Omron CX-Programmer project 新規ﾌﾟﾛｼﾞｪｸﾄ (CX-Programmer 9.61)

# PLC hoge1: CP1L L

## Program 新規ﾌﾟﾛｸﾞﾗﾑ1 (cyclic task 0)
Local symbols
I 0.00 BOOL
Q 100.00 BOOL

### Section ｾｸｼｮﾝ1

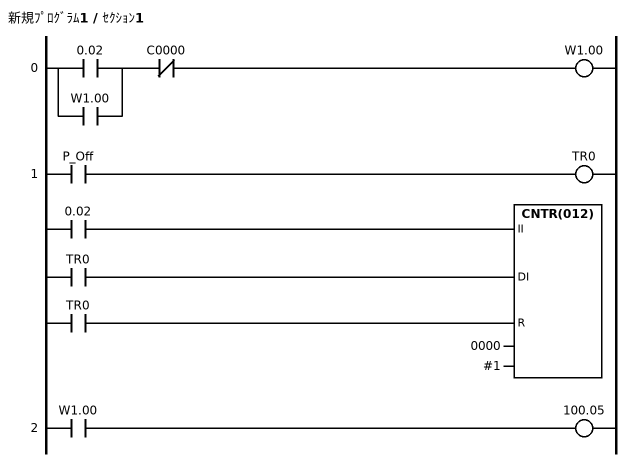
; rung 0
LD 0.02
OR W1.00
ANDNOT C0000
OUT W1.00
; rung 1
LD 0.02
LD P_Off
OUT TR0
LD TR0
CNTR(012) 0000 #1
; rung 2
LD W1.00
OUT 100.05

### Section END
; rung 0
END(001)